(*

short summary
=============

.. <legal notes>

legal notes
=================
| SPDX-FileCopyrightText: © 2023 ekvip automation GmbH <info@ekvip.de>
| SPDX-License-Identifier: Apache-2.0
| For details check: Apache-2.0_

.. _Apache-2.0: https://www.apache.org/licenses/LICENSE-2.0

.. </legal notes>

*)

{warning 'header is generated please add your documentation'}
TYPE containsDataStr :
STRUCT
	StringToTest		: STRING;
	WStringToTest 		: WSTRING;
	StringToContain 	: STRING;
	WStringToContain	: WSTRING;
	IgnoreCases			: BOOL;
	Trim 				: BOOL;
	ExpectedResult  	: BOOL;
	typeToTest      	: TypeToTest;		
END_STRUCT
END_TYPE

(* stored: Version 1.1.0.1, ProductVersion 3.1.4024.12
   DUT containsDataStr: Id {3cd23559-107f-4a5d-a883-48d18d3f3228} *)
